FUNCTION F_IncreaseTemperature

VAR_INPUT
	stMachine : REFERENCE TO ST_MachineOperatingParameters;
	tCycleTime : REAL;
END_VAR

VAR
END_VAR

stMachine.fTemperature := stMachine.fTemperature + (stMachine.fHeatingConstant * tCycleTime);

END_FUNCTION

(* stored: Version 1.1.0.1, ProductVersion 3.1.4024.12
   POU F_IncreaseTemperature: Id {89493a0d-ce5a-49fa-90a2-aaa7c6e5a758}, SpecialFunc None *)
